// TwinCAT 3 PLC project Fraktal_Press_Demo
// Title: Fraktal_Press_Demo
// Company: fraktal-automation
// Author: fraktal-automation
// ProjectVersion: 0.1.0.9
// Description: CX2030 virtual/physical commissioning example: XTI-linked EK1200/EL1809/EL2809 HAL mapping, two-hand start, interlocked door/part slide, safety aliases, Control On/Off, AUTO/HOME/MANUAL, and model recipes.
// ProgramVersion: 3.1.4026.24
// libraries:
//   Fraktal_Core, 0.1.0.5 (fraktal-automation)
//   Fraktal_Modules, 0.1.0.4 (fraktal-automation)
//   Tc2_EtherCAT, * (Beckhoff Automation GmbH)
//   Tc2_Standard, * (Beckhoff Automation GmbH)
//   Tc2_System, * (Beckhoff Automation GmbH)
//   Tc3_Module, * (Beckhoff Automation GmbH)
// project tree:
//   00_System/Hardware/ GVL_PressIO.TcGVL, GVL_PressSafety.TcGVL (not stored)
//   / PlcTask.TcTTO (not stored)
//   01_PneumaticPress/Sequences/ FB_PressDemoLoadPosition.TcPOU, FB_PressDemoHome.TcPOU, FB_PressDemoChangeover.TcPOU, FB_PressDemoAuto.TcPOU
//   01_PneumaticPress/Release/ FB_PressDemoRelease.TcPOU (not stored)
//   01_PneumaticPress/ FB_PressDemoUnit.TcPOU
//   00_System/ MAIN.TcPOU, FB_PressIoDriver.TcPOU, FB_PressControlOnCircuit.TcPOU, FB_PressControlDomain.TcPOU, FB_PressOutputAuthority.TcPOU (not stored), FB_PressSimulationDriver.TcPOU (not stored)
//   01_PneumaticPress/Recipes/ FB_PressRecipeCatalog.TcPOU (not stored)
//   01_PneumaticPress/Io/ FB_PressIoCatalog.TcPOU (not stored), GVL_PressFieldbus.TcGVL (not stored)
// real-time tasks:
//   TASK PlcTask: cycle T#10ms, priority 20, ADS port 350
// I/O:
//   DEVICE =000+S-A610-A1 (EtherCAT), AmsNetId 0.0.0.0.2.1
//     =000+S-K010 (EK1200) [EK1200-5000 EtherCAT Power supply (2A E-Bus)]
//       =000+S-K010B1 (EL1809) [EL1809 16Ch. Dig. Input 24V, 3ms]
//       =000+S-K010C1 (EL2809) [EL2809 16Ch. Dig. Output 24V, 0.5A]
//       =000+S-K010D1 (EL6001) [EL6001 Interface (RS232)]
//       =000+S-K010E (EL9011) [EL9011 End Terminal]
// variable links:
//   Fraktal_Press_Demo/Fraktal_Press_Demo Instance <-> =000+S-A610-A1 (EtherCAT)/=000+S-K010 (EK1200)/=000+S-K010B1 (EL1809)
//     PlcTask Inputs/GVL_PressIO._000K910A <-> Channel 15/_000K910A
//     PlcTask Inputs/GVL_PressIO._000K911_Y32 <-> Channel 14/_000K911_Y32
//     PlcTask Inputs/GVL_PressIO._000MB085A_2 <-> Channel 10/_000MB085A_2
//     PlcTask Inputs/GVL_PressIO._000MB085A_4 <-> Channel 11/_000MB085A_4
//     PlcTask Inputs/GVL_PressIO._101B201A <-> Channel 3/_101B201A
//     PlcTask Inputs/GVL_PressIO._101B202A <-> Channel 5/_101B202A
//     PlcTask Inputs/GVL_PressIO._101B301A <-> Channel 1/_101B301A
//     PlcTask Inputs/GVL_PressIO._101B201B <-> Channel 4/_101B201B
//     PlcTask Inputs/GVL_PressIO._101B202B <-> Channel 6/_101B202B
//     PlcTask Inputs/GVL_PressIO._101B301B <-> Channel 2/_101B301B
//     PlcTask Inputs/GVL_PressIO._101B601 <-> Channel 12/_101B601
//     PlcTask Inputs/GVL_PressIO._101S101 <-> Channel 7/_101S101
//     PlcTask Inputs/GVL_PressIO._101S102 <-> Channel 8/_101S102
//   Fraktal_Press_Demo/Fraktal_Press_Demo Instance <-> =000+S-A610-A1 (EtherCAT)/=000+S-K010 (EK1200)/=000+S-K010C1 (EL2809)
//     PlcTask Outputs/GVL_PressIO._000K911_A1 <-> Channel 11/_000K911_A1
//     PlcTask Outputs/GVL_PressIO._000K951_A1 <-> Channel 10/_000K951_A1
//     PlcTask Outputs/GVL_PressIO._101K201A <-> Channel 3/_101K201A
//     PlcTask Outputs/GVL_PressIO._101K202A <-> Channel 5/_101K202A
//     PlcTask Outputs/GVL_PressIO._101K301A <-> Channel 1/_101K301A
//     PlcTask Outputs/GVL_PressIO._101K201B <-> Channel 4/_101K201B
//     PlcTask Outputs/GVL_PressIO._101K202B <-> Channel 6/_101K202B
//     PlcTask Outputs/GVL_PressIO._101K301B <-> Channel 2/_101K301B
//     PlcTask Outputs/GVL_PressIO._101P101 <-> Channel 7/_101P101
//     PlcTask Outputs/GVL_PressIO._101P102 <-> Channel 8/_101P102

// ---- 00_System/Hardware/GVL_PressIO.TcGVL
{attribute 'qualified_only'}
// CX2030 local EtherCAT process image, reconciled with the supplied XTI export.
// TcLinkTo owns the physical link by exact terminal/channel/PDO-entry name;
// AT %I*/%Q* keeps the compiler-selected process-image offset non-positional.
VAR_GLOBAL
    // =000+S-K010B1 (EL1809) inputs
    {attribute 'TcLinkTo' := 'TIIB[=000+S-K010B1 (EL1809)]^Channel 1^_101B301A'}
    _101B301A AT %I* : BOOL;       // Ch1 feeder retracted = logical slide INSIDE
    {attribute 'TcLinkTo' := 'TIIB[=000+S-K010B1 (EL1809)]^Channel 2^_101B301B'}
    _101B301B AT %I* : BOOL;       // Ch2 feeder extended  = logical slide OUTSIDE
    {attribute 'TcLinkTo' := 'TIIB[=000+S-K010B1 (EL1809)]^Channel 3^_101B201A'}
    _101B201A AT %I* : BOOL;       // Ch3 door closed
    {attribute 'TcLinkTo' := 'TIIB[=000+S-K010B1 (EL1809)]^Channel 4^_101B201B'}
    _101B201B AT %I* : BOOL;       // Ch4 door open
    {attribute 'TcLinkTo' := 'TIIB[=000+S-K010B1 (EL1809)]^Channel 5^_101B202A'}
    _101B202A AT %I* : BOOL;       // Ch5 press down
    {attribute 'TcLinkTo' := 'TIIB[=000+S-K010B1 (EL1809)]^Channel 6^_101B202B'}
    _101B202B AT %I* : BOOL;       // Ch6 press up
    {attribute 'TcLinkTo' := 'TIIB[=000+S-K010B1 (EL1809)]^Channel 7^_101S101'}
    _101S101  AT %I* : BOOL;       // Ch7 right two-hand raw button
    {attribute 'TcLinkTo' := 'TIIB[=000+S-K010B1 (EL1809)]^Channel 8^_101S102'}
    _101S102  AT %I* : BOOL;       // Ch8 left two-hand raw button
    {attribute 'TcLinkTo' := 'TIIB[=000+S-K010B1 (EL1809)]^Channel 10^_000MB085A_2'}
    _000MB085A_2 AT %I* : BOOL;    // Ch10 compressed air below 0.3 bar
    {attribute 'TcLinkTo' := 'TIIB[=000+S-K010B1 (EL1809)]^Channel 11^_000MB085A_4'}
    _000MB085A_4 AT %I* : BOOL;    // Ch11 compressed air above 4.5 bar
    {attribute 'TcLinkTo' := 'TIIB[=000+S-K010B1 (EL1809)]^Channel 12^_101B601'}
    _101B601 AT %I* : BOOL;        // Ch12 part present
    // N54 D2 operator buttons. Free EL1809 channels were 9/13/16; 9 and 13 are
    // assigned here. The TcLinkTo names MUST match the terminal channel names in
    // XAE - confirm the physical wiring before trusting these.
    {attribute 'TcLinkTo' := 'TIIB[=000+S-K010B1 (EL1809)]^Channel 9^_000BS901'}
    _000BS901 AT %I* : BOOL;       // Ch9  IsControlOnButtonPressed  (=000+B-S901:14)
    {attribute 'TcLinkTo' := 'TIIB[=000+S-K010B1 (EL1809)]^Channel 13^_000BS902'}
    _000BS902 AT %I* : BOOL;       // Ch13 IsControlOffButtonPressed (=000+B-S902:14)
    {attribute 'TcLinkTo' := 'TIIB[=000+S-K010B1 (EL1809)]^Channel 14^_000K911_Y32'}
    _000K911_Y32 AT %I* : BOOL;    // Ch14 Control On feedback
    {attribute 'TcLinkTo' := 'TIIB[=000+S-K010B1 (EL1809)]^Channel 15^_000K910A'}
    _000K910A AT %I* : BOOL;       // Ch15 E-stop PRESSED (=000+S1-K910A:14); NORMALLY OPEN on this
                                   // demo rig: TRUE = actuated. NOT fail-safe - production needs NC.

    // =000+S-K010C1 (EL2809) outputs
    {attribute 'TcLinkTo' := 'TIIB[=000+S-K010C1 (EL2809)]^Channel 1^_101K301A'}
    _101K301A AT %Q* : BOOL;       // Ch1 feeder backward = move inside
    {attribute 'TcLinkTo' := 'TIIB[=000+S-K010C1 (EL2809)]^Channel 2^_101K301B'}
    _101K301B AT %Q* : BOOL;       // Ch2 feeder forward  = move outside
    {attribute 'TcLinkTo' := 'TIIB[=000+S-K010C1 (EL2809)]^Channel 3^_101K201A'}
    _101K201A AT %Q* : BOOL;       // Ch3 close door
    {attribute 'TcLinkTo' := 'TIIB[=000+S-K010C1 (EL2809)]^Channel 4^_101K201B'}
    _101K201B AT %Q* : BOOL;       // Ch4 open door
    {attribute 'TcLinkTo' := 'TIIB[=000+S-K010C1 (EL2809)]^Channel 5^_101K202A'}
    _101K202A AT %Q* : BOOL;       // Ch5 press downward
    {attribute 'TcLinkTo' := 'TIIB[=000+S-K010C1 (EL2809)]^Channel 6^_101K202B'}
    _101K202B AT %Q* : BOOL;       // Ch6 press upward
    {attribute 'TcLinkTo' := 'TIIB[=000+S-K010C1 (EL2809)]^Channel 7^_101P101'}
    _101P101  AT %Q* : BOOL;       // Ch7 right two-hand lamp
    {attribute 'TcLinkTo' := 'TIIB[=000+S-K010C1 (EL2809)]^Channel 8^_101P102'}
    _101P102  AT %Q* : BOOL;       // Ch8 left two-hand lamp
    {attribute 'TcLinkTo' := 'TIIB[=000+S-K010C1 (EL2809)]^Channel 10^_000K951_A1'}
    _000K951_A1 AT %Q* : BOOL;     // Ch10 SwitchControlOn functional request
    {attribute 'TcLinkTo' := 'TIIB[=000+S-K010C1 (EL2809)]^Channel 11^_000K911_A1'}
    _000K911_A1 AT %Q* : BOOL;     // Ch11 EnableControlOn functional request
END_VAR

// ---- 01_PneumaticPress/Sequences/FB_PressDemoLoadPosition.TcPOU
// Shared load-safe-position sub-sequence (Core §6.7): ram up, door open, slide
// outside. HOME and CHANGEOVER both embed it as one composite step, passing a
// BaseStepNo window so its detailed progress projects through the Unit's normal
// §6.5 step record. Implemented as a Core §6.8 ST `CASE _step OF` skeleton on
// FB_SequenceBase — the step actions issue child commands only through the §6.1
// handshake (M_MayIssue), and progression rides the shared _retVal via M_Advance.
FUNCTION_BLOCK FB_PressDemoLoadPosition EXTENDS FB_SequenceBase
VAR
    _baseStepNo : INT;
    {attribute 'OPC.UA.DA' := '0'}
    _pressRam : REFERENCE TO FB_CylinderCM;
    {attribute 'OPC.UA.DA' := '0'}
    _door : REFERENCE TO FB_CylinderCM;
    {attribute 'OPC.UA.DA' := '0'}
    _partSlide : REFERENCE TO FB_CylinderCM;
END_VAR

// step body runs via M_Run; the Unit calls this instance each scan

METHOD M_Reset
VAR_INPUT
    BaseStepNo : INT;
END_VAR
_baseStepNo := BaseStepNo;
M_ResetBase();
END_METHOD

// §6.8 ST step skeleton. One M_Step per step, one commit via M_Advance.
METHOD M_Run
IF NOT _attached THEN
    RETURN;
END_IF
CASE _step OF
    0:  // ram up
        M_Step(StepNo := _baseStepNo, StepName := 'project.step.pressSafePositionRamUp',
            Awaits := _pressRam, AwaitingLabel := 'PressRam.RETRACT',
            TimeClass := E_TimeClass.WORK, ExpectedTime := T#0S);
        IF M_MayIssue(Steppable := TRUE) THEN
            _pressRam.Abort := FALSE;
            _pressRam.Command := E_CylinderCommand.RETRACT;
            _pressRam.Execute := TRUE;
        END_IF
        IF _pressRam.Done THEN
            _pressRam.Execute := FALSE;
            _retVal := E_StepResult.ADVANCE;
        END_IF
        M_Advance(OnAdvance := 20);
    20:  // door open
        M_Step(StepNo := _baseStepNo + 20, StepName := 'project.step.pressSafePositionDoorOpen',
            Awaits := _door, AwaitingLabel := 'Door.RETRACT',
            TimeClass := E_TimeClass.WORK, ExpectedTime := T#0S);
        IF M_MayIssue(Steppable := TRUE) THEN
            _door.Abort := FALSE;
            _door.Command := E_CylinderCommand.RETRACT;
            _door.Execute := TRUE;
        END_IF
        IF _door.Done THEN
            _door.Execute := FALSE;
            _retVal := E_StepResult.ADVANCE;
        END_IF
        M_Advance(OnAdvance := 40);
    40:  // slide outside
        M_Step(StepNo := _baseStepNo + 40, StepName := 'project.step.pressSafePositionSlideOutside',
            Awaits := _partSlide, AwaitingLabel := 'PartSlide.RETRACT',
            TimeClass := E_TimeClass.WORK, ExpectedTime := T#0S);
        IF M_MayIssue(Steppable := TRUE) THEN
            _partSlide.Abort := FALSE;
            _partSlide.Command := E_CylinderCommand.RETRACT;
            _partSlide.Execute := TRUE;
        END_IF
        IF _partSlide.Done THEN
            _partSlide.Execute := FALSE;
            _retVal := E_StepResult.ADVANCE;
        END_IF
        M_Advance(OnAdvance := 999);
    999:  // established
        M_Step(StepNo := _baseStepNo + 60, StepName := 'project.step.pressSafePositionComplete',
            Awaits := 0, AwaitingLabel := '', TimeClass := E_TimeClass.WORK, ExpectedTime := T#0S);
        Done := TRUE;
ELSE
    M_Fault(Reason := E_Reason.STEP_STALLED, DescriptionKey := 'std.error.undefinedStep');
END_CASE
END_METHOD

METHOD Setup : BOOL
VAR_INPUT
    Host : I_SequenceHost;
END_VAR
VAR_IN_OUT
    PressRam : FB_CylinderCM;
    Door : FB_CylinderCM;
    PartSlide : FB_CylinderCM;
END_VAR
_pressRam REF= PressRam;
_door REF= Door;
_partSlide REF= PartSlide;
Setup := M_Attach(Host := Host)
    AND __ISVALIDREF(_pressRam) AND __ISVALIDREF(_door) AND __ISVALIDREF(_partSlide);
END_METHOD

END_FUNCTION_BLOCK

// ---- 01_PneumaticPress/Sequences/FB_PressDemoHome.TcPOU
// HOME mode chain (Core §6.2/§6.8 ST skeleton on FB_SequenceBase): establish the
// shared load-safe position, then complete. Finite (does not loop).
FUNCTION_BLOCK FB_PressDemoHome EXTENDS FB_SequenceBase
VAR
    {attribute 'OPC.UA.DA' := '0'}
    _outCmd : REFERENCE TO ST_PneumaticPressOutCmd;
    {attribute 'OPC.UA.DA' := '0'}
    _loadPosition : FB_PressDemoLoadPosition;
    _loadPositionRunning : BOOL;
END_VAR

METHOD M_Reset
M_ResetBase();
_loadPositionRunning := FALSE;
_loadPosition.M_Reset(BaseStepNo := 0);
END_METHOD

METHOD M_Run
IF NOT _attached THEN
    RETURN;
END_IF
CASE _step OF
    0:  // initialize
        M_Step(StepNo := 0, StepName := 'project.step.pressHomeInitialize',
            Awaits := 0, AwaitingLabel := '', TimeClass := E_TimeClass.WORK, ExpectedTime := T#0S);
        _outCmd.Homed := FALSE;
        _outCmd.ChangeoverCompleted := FALSE;
        _loadPositionRunning := FALSE;
        _retVal := E_StepResult.ADVANCE;
        M_Advance(OnAdvance := 900);
    900:  // shared load-safe position (composite step, §6.7)
        IF NOT _loadPositionRunning THEN
            _loadPosition.M_Reset(BaseStepNo := 900);
            _loadPositionRunning := TRUE;
        END_IF
        _loadPosition.M_Run();
        IF _loadPosition.Done THEN
            _loadPositionRunning := FALSE;
            _retVal := E_StepResult.ADVANCE;
        END_IF
        M_Advance(OnAdvance := 999);
    999:  // complete
        M_Step(StepNo := 999, StepName := 'project.step.pressHomeComplete',
            Awaits := 0, AwaitingLabel := '', TimeClass := E_TimeClass.WORK, ExpectedTime := T#0S);
        _outCmd.Homed := TRUE;
        M_Complete();
ELSE
    M_Fault(Reason := E_Reason.STEP_STALLED, DescriptionKey := 'std.error.undefinedStep');
END_CASE
END_METHOD

METHOD Setup : BOOL
VAR_INPUT
    Host : I_SequenceHost;
END_VAR
VAR_IN_OUT
    PressRam : FB_CylinderCM;
    Door : FB_CylinderCM;
    PartSlide : FB_CylinderCM;
    OutCmd : ST_PneumaticPressOutCmd;
END_VAR
_outCmd REF= OutCmd;
Setup := M_Attach(Host := Host) AND __ISVALIDREF(_outCmd)
    AND _loadPosition.Setup(Host := Host, PressRam := PressRam, Door := Door, PartSlide := PartSlide);
END_METHOD

END_FUNCTION_BLOCK

// ---- 01_PneumaticPress/Sequences/FB_PressDemoChangeover.TcPOU
// CHANGEOVER mode chain (Core §6.2/§6.8 ST skeleton on FB_SequenceBase): validate
// the selected model, establish the shared load-safe position, then ask the
// operator (§6.11) to confirm tooling/material match before completing. The
// 'repeat position' answer restarts the guided move via a backward jump (§6.10).
FUNCTION_BLOCK FB_PressDemoChangeover EXTENDS FB_SequenceBase
VAR
    _decisionRequest : ST_DecisionRequest;
    _answer : INT;
    _modelSelected : BOOL;
    {attribute 'OPC.UA.DA' := '0'}
    _outCmd : REFERENCE TO ST_PneumaticPressOutCmd;
    {attribute 'OPC.UA.DA' := '0'}
    _model : REFERENCE TO ST_ModelId;
    {attribute 'OPC.UA.DA' := '0'}
    _loadPosition : FB_PressDemoLoadPosition;
    _loadPositionRunning : BOOL;
END_VAR

METHOD M_Reset
M_ResetBase();
_answer := 0;
_loadPositionRunning := FALSE;
_loadPosition.M_Reset(BaseStepNo := 0);
END_METHOD

METHOD M_Run
IF NOT _attached THEN
    RETURN;
END_IF
CASE _step OF
    0:  // initialize
        M_Step(StepNo := 0, StepName := 'project.step.pressChangeoverInitialize',
            Awaits := 0, AwaitingLabel := '', TimeClass := E_TimeClass.WORK, ExpectedTime := T#0S);
        _outCmd.ChangeoverCompleted := FALSE;
        _outCmd.Homed := FALSE;
        _answer := 0;
        _decisionRequest.Prompt := '';
        M_ClearDecision();
        _loadPositionRunning := FALSE;
        _retVal := E_StepResult.ADVANCE;
        M_Advance(OnAdvance := 800);
    800:  // validate the transactionally-loaded model
        M_Step(StepNo := 800, StepName := 'project.step.pressChangeoverValidateModel',
            Awaits := 0, AwaitingLabel := '', TimeClass := E_TimeClass.WAIT_OPERATOR, ExpectedTime := T#0S);
        _modelSelected := M_Await(Idx := 1, Label := 'project.condition.pressModelSelected',
            Ok := _model.ModelCode <> '');
        IF _modelSelected THEN
            _loadPositionRunning := FALSE;
            _retVal := E_StepResult.ADVANCE;
        END_IF
        M_Advance(OnAdvance := 810);
    810:  // shared load-safe position (composite step)
        IF NOT _loadPositionRunning THEN
            _loadPosition.M_Reset(BaseStepNo := 810);
            _loadPositionRunning := TRUE;
        END_IF
        _loadPosition.M_Run();
        IF _loadPosition.Done THEN
            _loadPositionRunning := FALSE;
            _retVal := E_StepResult.ADVANCE;
        END_IF
        M_Advance(OnAdvance := 870);
    870:  // request tooling/material confirmation
        M_Step(StepNo := 870, StepName := 'project.step.pressChangeoverRequestConfirmation',
            Awaits := 0, AwaitingLabel := '', TimeClass := E_TimeClass.WAIT_OPERATOR, ExpectedTime := T#0S);
        _decisionRequest.Prompt := 'project.decision.pressChangeoverConfirm';
        _decisionRequest.Options[1] := 'project.decision.confirmChangeover';
        _decisionRequest.Options[2] := 'project.decision.repeatChangeoverPosition';
        _decisionRequest.Default := 0;
        _decisionRequest.Timeout := T#0S;
        M_AskDecision(Req := _decisionRequest);
        _retVal := E_StepResult.ADVANCE;
        M_Advance(OnAdvance := 880);
    880:  // await confirmation; JUMP1 = repeat the guided position
        M_Step(StepNo := 880, StepName := 'project.step.pressChangeoverAwaitConfirmation',
            Awaits := 0, AwaitingLabel := '', TimeClass := E_TimeClass.WAIT_OPERATOR, ExpectedTime := T#0S);
        _answer := M_TakeDecision();
        IF _answer = 1 THEN
            _retVal := E_StepResult.ADVANCE;
        ELSIF _answer = 2 THEN
            _loadPositionRunning := FALSE;      // repeat the guided position from the start
            _retVal := E_StepResult.JUMP1;
        ELSE
            _modelSelected := M_Await(Idx := 1,
                Label := 'project.condition.pressChangeoverConfirmation', Ok := FALSE);
        END_IF
        M_Advance(OnAdvance := 999, OnJump1 := 810);
    999:  // complete
        M_Step(StepNo := 999, StepName := 'project.step.pressChangeoverComplete',
            Awaits := 0, AwaitingLabel := '', TimeClass := E_TimeClass.WORK, ExpectedTime := T#0S);
        _outCmd.Homed := TRUE;
        _outCmd.ChangeoverCompleted := TRUE;
        M_Complete();
ELSE
    M_Fault(Reason := E_Reason.STEP_STALLED, DescriptionKey := 'std.error.undefinedStep');
END_CASE
END_METHOD

METHOD Setup : BOOL
VAR_INPUT
    Host : I_SequenceHost;
END_VAR
VAR_IN_OUT
    PressRam : FB_CylinderCM;
    Door : FB_CylinderCM;
    PartSlide : FB_CylinderCM;
    OutCmd : ST_PneumaticPressOutCmd;
    Model : ST_ModelId;
END_VAR
_outCmd REF= OutCmd;
_model REF= Model;
Setup := M_Attach(Host := Host) AND __ISVALIDREF(_outCmd) AND __ISVALIDREF(_model)
    AND _loadPosition.Setup(Host := Host, PressRam := PressRam, Door := Door, PartSlide := PartSlide);
END_METHOD

END_FUNCTION_BLOCK

// ---- 01_PneumaticPress/Sequences/FB_PressDemoAuto.TcPOU
// AUTO mode chain (Core §6.2/§6.8 ST skeleton on FB_SequenceBase): the continuous
// production cycle — await a fresh two-hand start with part+air present, transfer
// the part in, press for the recipe dwell, return to load position, count the good
// part, and loop until Stop. A Stop requested at the between-cycles wait is honored
// there (M_StopNow) so no phantom cycle is charged. Every child motion goes through
// the §6.1 handshake (M_MayIssue); progression rides the shared _retVal.
FUNCTION_BLOCK FB_PressDemoAuto EXTENDS FB_SequenceBase
VAR
    _partReady, _airReady, _startReady : BOOL;
    _traceAccepted, _recordAccepted, _partProcessed : BOOL;
    {attribute 'OPC.UA.DA' := '0'}
    _pressRam : REFERENCE TO FB_CylinderCM;
    {attribute 'OPC.UA.DA' := '0'}
    _door : REFERENCE TO FB_CylinderCM;
    {attribute 'OPC.UA.DA' := '0'}
    _partSlide : REFERENCE TO FB_CylinderCM;
    {attribute 'OPC.UA.DA' := '0'}
    _twoHand : REFERENCE TO FB_TwoHandStartCM;
    {attribute 'OPC.UA.DA' := '0'}
    _partPresentSensor : REFERENCE TO FB_DigitalInputCM;
    {attribute 'OPC.UA.DA' := '0'}
    _airPressureMonitor : REFERENCE TO FB_AirPressureMonitorCM;
    {attribute 'OPC.UA.DA' := '0'}
    _parCfg : REFERENCE TO ST_PneumaticPressParCfg;
    {attribute 'OPC.UA.DA' := '0'}
    _outCmd : REFERENCE TO ST_PneumaticPressOutCmd;
    {attribute 'OPC.UA.DA' := '0'}
    _startLatched : REFERENCE TO BOOL;
    {attribute 'OPC.UA.DA' := '0'}
    _loadPosition : FB_PressDemoLoadPosition;
    _loadPositionRunning : BOOL;
END_VAR

METHOD M_Reset
M_ResetBase(0);
_loadPositionRunning := FALSE;
_loadPosition.M_Reset(BaseStepNo := 0);
END_METHOD

METHOD M_Run
IF NOT _attached THEN
    RETURN;
END_IF
CASE _step OF
    0:  // initialize
        M_Step(StepNo := 0, StepName := 'project.step.pressAutoInitialize',
            Awaits := 0, AwaitingLabel := '', TimeClass := E_TimeClass.WORK, ExpectedTime := T#0S);
        _outCmd.CycleCompleted := FALSE;
        _outCmd.Homed := FALSE;
        _outCmd.ChangeoverCompleted := FALSE;
        _loadPositionRunning := FALSE;
        _retVal := E_StepResult.ADVANCE;
        M_Advance(OnAdvance := 100, OnJump1 := -1, OnJump2 := -1, OnJump3 := -1);
    100:  // await a fresh two-hand start (the §8.11.1 cycle-start marker)
        M_Step(StepNo := 100, StepName := 'project.step.pressAwaitTwoHand',
            Awaits := 0, AwaitingLabel := '', TimeClass := E_TimeClass.WAIT_OPERATOR, ExpectedTime := T#0S);
        _outCmd.CycleCompleted := FALSE;
        _partReady := M_Await(Idx := 1, Label := 'project.condition.partPresent',
            Ok := _partPresentSensor.OutImm.Value AND _partPresentSensor.OutImm.Quality);
        _airReady := M_Await(Idx := 2, Label := 'project.condition.airPressureOk',
            Ok := _airPressureMonitor.OutImm.PressureOk);
        IF _parCfg.RequireTwoHandStart THEN
            _startReady := M_Await(Idx := 3, Label := 'project.condition.twoHandStart', Ok := _startLatched);
        ELSE
            _startReady := TRUE;
        END_IF
        IF M_StopPending() THEN
            M_StopNow();                       // stop accepted BETWEEN cycles: no phantom cycle
        ELSIF _partReady AND _airReady AND _startReady THEN
            _traceAccepted := M_PartReceived();
            _retVal := E_StepResult.ADVANCE;
        END_IF
        M_Advance(OnAdvance := 110, OnJump1 := -1, OnJump2 := -1, OnJump3 := -1);
    110:  // ram up
        M_Step(StepNo := 110, StepName := 'project.step.pressRamUp',
            Awaits := _pressRam, AwaitingLabel := 'PressRam.RETRACT', TimeClass := E_TimeClass.WORK, ExpectedTime := T#0S);
        IF M_MayIssue(Steppable := TRUE) THEN
            _pressRam.Abort := FALSE; _pressRam.Command := E_CylinderCommand.RETRACT; _pressRam.Execute := TRUE;
        END_IF
        IF _pressRam.Done THEN _pressRam.Execute := FALSE; _retVal := E_StepResult.ADVANCE; END_IF
        M_Advance(OnAdvance := 130, OnJump1 := -1, OnJump2 := -1, OnJump3 := -1);
    130:  // door open
        M_Step(StepNo := 130, StepName := 'project.step.pressDoorOpen',
            Awaits := _door, AwaitingLabel := 'Door.RETRACT', TimeClass := E_TimeClass.WORK, ExpectedTime := T#0S);
        IF M_MayIssue(Steppable := TRUE) THEN
            _door.Abort := FALSE; _door.Command := E_CylinderCommand.RETRACT; _door.Execute := TRUE;
        END_IF
        IF _door.Done THEN _door.Execute := FALSE; _retVal := E_StepResult.ADVANCE; END_IF
        M_Advance(OnAdvance := 150, OnJump1 := -1, OnJump2 := -1, OnJump3 := -1);
    150:  // slide inside (value-adding sequence begins)
        M_Step(StepNo := 150, StepName := 'project.step.pressSlideInside',
            Awaits := _partSlide, AwaitingLabel := 'PartSlide.EXTEND', TimeClass := E_TimeClass.WORK, ExpectedTime := T#0S);
        IF M_MayIssue(Steppable := TRUE) THEN
            M_PartStarted();
            _partSlide.Abort := FALSE; _partSlide.Command := E_CylinderCommand.EXTEND; _partSlide.Execute := TRUE;
        END_IF
        IF _partSlide.Done THEN _partSlide.Execute := FALSE; _retVal := E_StepResult.ADVANCE; END_IF
        M_Advance(OnAdvance := 170, OnJump1 := -1, OnJump2 := -1, OnJump3 := -1);
    170:  // transfer settle
        M_Step(StepNo := 170, StepName := 'project.step.pressTransferSettle',
            Awaits := 0, AwaitingLabel := '', TimeClass := E_TimeClass.WORK, ExpectedTime := _parCfg.TransferSettleTime);
        _retVal := M_Delay(PT := _parCfg.TransferSettleTime);
        M_Advance(OnAdvance := 180, OnJump1 := -1, OnJump2 := -1, OnJump3 := -1);
    180:  // door close
        M_Step(StepNo := 180, StepName := 'project.step.pressDoorClose',
            Awaits := _door, AwaitingLabel := 'Door.EXTEND', TimeClass := E_TimeClass.WORK, ExpectedTime := T#0S);
        IF M_MayIssue(Steppable := TRUE) THEN
            _door.Abort := FALSE; _door.Command := E_CylinderCommand.EXTEND; _door.Execute := TRUE;
        END_IF
        IF _door.Done THEN _door.Execute := FALSE; _retVal := E_StepResult.ADVANCE; END_IF
        M_Advance(OnAdvance := 200, OnJump1 := -1, OnJump2 := -1, OnJump3 := -1);
    200:  // ram down
        M_Step(StepNo := 200, StepName := 'project.step.pressRamDown',
            Awaits := _pressRam, AwaitingLabel := 'PressRam.EXTEND', TimeClass := E_TimeClass.WORK, ExpectedTime := T#0S);
        IF M_MayIssue(Steppable := TRUE) THEN
            _pressRam.Abort := FALSE; _pressRam.Command := E_CylinderCommand.EXTEND; _pressRam.Execute := TRUE;
        END_IF
        IF _pressRam.Done THEN _pressRam.Execute := FALSE; _retVal := E_StepResult.ADVANCE; END_IF
        M_Advance(OnAdvance := 220, OnJump1 := -1, OnJump2 := -1, OnJump3 := -1);
    220:  // press dwell — two-hand must stay active
        M_Step(StepNo := 220, StepName := 'project.step.pressDwell',
            Awaits := 0, AwaitingLabel := '', TimeClass := E_TimeClass.WORK, ExpectedTime := _parCfg.PressSettleTime);
        IF NOT _twoHand.OutImm.SafeActive AND _parCfg.RequireTwoHandStart THEN
            _pressRam.WithdrawOutputs();
            M_Fault(Reason := E_Reason.INTERLOCK_DROPPED, DescriptionKey := 'project.error.twoHandReleasedDuringPress');
        ELSE
            _retVal := M_Delay(PT := _parCfg.PressSettleTime);
        END_IF
        M_Advance(OnAdvance := 230, OnJump1 := -1, OnJump2 := -1, OnJump3 := -1);
    230:  // record the applied dwell (§3.16.1 measured value)
        M_Step(StepNo := 230, StepName := 'project.step.pressRecordResult',
            Awaits := 0, AwaitingLabel := '', TimeClass := E_TimeClass.WORK, ExpectedTime := T#0S);
        _recordAccepted := M_PartRecord(RecordName := 'PressDwell',
            Value := DINT_TO_LREAL(TIME_TO_DINT(_parCfg.PressSettleTime)),
            Minimum := 0, Maximum := 30000,
            Target := DINT_TO_LREAL(TIME_TO_DINT(_parCfg.PressSettleTime)), EngUnit := 'ms');
        _loadPositionRunning := FALSE;
        _retVal := E_StepResult.ADVANCE;
        M_Advance(OnAdvance := 240, OnJump1 := -1, OnJump2 := -1, OnJump3 := -1);
    240:  // return to the shared load-safe position (composite step)
        IF NOT _loadPositionRunning THEN
            _loadPosition.M_Reset(BaseStepNo := 240);
            _loadPositionRunning := TRUE;
        END_IF
        _loadPosition.M_Run();
        IF _loadPosition.Done THEN
            _loadPositionRunning := FALSE;
            _retVal := E_StepResult.ADVANCE;
        END_IF
        M_Advance(OnAdvance := 999, OnJump1 := -1, OnJump2 := -1, OnJump3 := -1);
    999:  // cycle complete — write result, count by verdict, loop (§8.11.1 finish marker)
        M_Step(StepNo := 999, StepName := 'project.step.pressAutoComplete',
            Awaits := 0, AwaitingLabel := '', TimeClass := E_TimeClass.WORK, ExpectedTime := T#0S);
        _outCmd.CycleCompleted := TRUE;
        _partProcessed := M_PartProcessed(Verdict := E_Verdict.OK, Reason := E_Reason.NONE);
        IF NOT _partProcessed THEN
            M_CountGood();                     // §3.9: no carrier configured — count directly
        END_IF
        _startLatched := FALSE;
        IF M_EndOfCycle() THEN
            _retVal := E_StepResult.ADVANCE;   // stop NOT requested: loop to N100
        END_IF
        M_Advance(OnAdvance := 100, OnJump1 := -1, OnJump2 := -1, OnJump3 := -1);
ELSE
    M_Fault(Reason := E_Reason.STEP_STALLED, DescriptionKey := 'std.error.undefinedStep');
END_CASE
END_METHOD

METHOD Setup : BOOL
VAR_INPUT
    Host : I_SequenceHost;
END_VAR
VAR_IN_OUT
    PressRam : FB_CylinderCM;
    Door : FB_CylinderCM;
    PartSlide : FB_CylinderCM;
    TwoHand : FB_TwoHandStartCM;
    PartPresentSensor : FB_DigitalInputCM;
    AirPressureMonitor : FB_AirPressureMonitorCM;
    ParCfg : ST_PneumaticPressParCfg;
    OutCmd : ST_PneumaticPressOutCmd;
    StartLatched : BOOL;
END_VAR
_pressRam REF= PressRam;
_door REF= Door;
_partSlide REF= PartSlide;
_twoHand REF= TwoHand;
_partPresentSensor REF= PartPresentSensor;
_airPressureMonitor REF= AirPressureMonitor;
_parCfg REF= ParCfg;
_outCmd REF= OutCmd;
_startLatched REF= StartLatched;
Setup := M_Attach(Host := Host) AND __ISVALIDREF(_pressRam) AND __ISVALIDREF(_door)
    AND __ISVALIDREF(_partSlide) AND __ISVALIDREF(_twoHand)
    AND __ISVALIDREF(_partPresentSensor) AND __ISVALIDREF(_airPressureMonitor)
    AND __ISVALIDREF(_parCfg) AND __ISVALIDREF(_outCmd) AND __ISVALIDREF(_startLatched)
    AND _loadPosition.Setup(Host := Host, PressRam := PressRam, Door := Door, PartSlide := PartSlide);
END_METHOD

END_FUNCTION_BLOCK

// ---- 01_PneumaticPress/FB_PressDemoUnit.TcPOU
// Project-owned Unit: pneumatic press + access door + transfer slide + two-hand request.
// Cylinder interlocks prevent the two documented collisions in AUTO and MANUAL.
// Certified E-stop, two-hand evaluation and safe valve outputs remain external.
FUNCTION_BLOCK FB_PressDemoUnit EXTENDS FB_UnitBase
VAR_INPUT
    ParCfg : ST_PneumaticPressParCfg;
    ParCmd : ST_PneumaticPressParCmd;
END_VAR
VAR_OUTPUT
    PressRam      : FB_CylinderCM;
    Door          : FB_CylinderCM;
    PartSlide     : FB_CylinderCM;
    TwoHand       : FB_TwoHandStartCM;
    PneumaticPower: FB_PowerGroupCM;
    PartPresentSensor : FB_DigitalInputCM;
    AirPressureMonitor : FB_AirPressureMonitorCM;
    ReleaseConditions : FB_PressDemoRelease; // project-owned, browseable condition state
    OutCmd        : ST_PneumaticPressOutCmd;
    OutImm        : ST_PneumaticPressOutImm;
END_VAR
VAR
    {attribute 'OPC.UA.DA' := '0'}
    _recipe : I_RecipeProvider;
    _parCfgStaged : ST_PneumaticPressParCfg;
    _recipePrepared : BOOL;
    _startLatched : BOOL;
    _powerRequestPending : BOOL;
    _powerTargetOn : BOOL;
    {attribute 'OPC.UA.DA' := '0'}
    _homeSequence : FB_PressDemoHome;       // §6.8 ST chain on FB_SequenceBase owns HOME steps
    {attribute 'OPC.UA.DA' := '0'}
    _changeoverSequence : FB_PressDemoChangeover;
    {attribute 'OPC.UA.DA' := '0'}
    _autoSequence : FB_PressDemoAuto;
END_VAR

Cyclic();

METHOD Setup : BOOL
VAR_INPUT
    Name : STRING(80);
    PressHal : REFERENCE TO ST_CylinderHal;
    DoorHal : REFERENCE TO ST_CylinderHal;
    SlideHal : REFERENCE TO ST_CylinderHal;
    TwoHandHal : REFERENCE TO ST_TwoHandHal;
    PowerHal : REFERENCE TO ST_PowerGroupHal;
    PartPresentHal : REFERENCE TO ST_DigitalInputHal;
    AirPressureHal : REFERENCE TO ST_AirPressureHal;
    Recipe : I_RecipeProvider;
END_VAR
VAR
    InitialModel : ST_ModelId;
    Ok : BOOL;
END_VAR
_M_SetName(Name);
_M_SetPresentation(DisplayNameKey := 'project.module.pneumaticPress.name', DescriptionKey := 'project.module.pneumaticPress.description');
_recipe := Recipe;
Ok := PressRam.Setup(Name := CONCAT(Name, '.PressRam'), HalRef := PressHal, Recipe := 0);
Ok := Door.Setup(Name := CONCAT(Name, '.Door'), HalRef := DoorHal, Recipe := 0) AND Ok;
Ok := PartSlide.Setup(Name := CONCAT(Name, '.PartSlide'), HalRef := SlideHal, Recipe := 0) AND Ok;
Ok := TwoHand.Setup(Name := CONCAT(Name, '.TwoHand'), HalRef := TwoHandHal) AND Ok;
Ok := PneumaticPower.Setup(Name := CONCAT(Name, '.PneumaticPower'), HalRef := PowerHal) AND Ok;
Ok := PartPresentSensor.Setup(Name := CONCAT(Name, '.PartPresentSensor'),
    HalRef := PartPresentHal, DisplayNameKey := 'project.module.partPresentSensor.name',
    DescriptionKey := 'project.module.partPresentSensor.description') AND Ok;
Ok := AirPressureMonitor.Setup(Name := CONCAT(Name, '.AirPressureMonitor'),
    HalRef := AirPressureHal) AND Ok;
Ok := ReleaseConditions.Setup(UnitPath := Name) AND Ok;
Ok := _homeSequence.Setup(Host := THIS^, PressRam := PressRam, Door := Door,
    PartSlide := PartSlide, OutCmd := OutCmd) AND Ok;
Ok := _changeoverSequence.Setup(Host := THIS^, PressRam := PressRam, Door := Door,
    PartSlide := PartSlide, OutCmd := OutCmd, Model := Model) AND Ok;
Ok := _autoSequence.Setup(Host := THIS^, PressRam := PressRam, Door := Door,
    PartSlide := PartSlide, TwoHand := TwoHand, PartPresentSensor := PartPresentSensor,
    AirPressureMonitor := AirPressureMonitor, ParCfg := ParCfg, OutCmd := OutCmd,
    StartLatched := _startLatched) AND Ok;
PneumaticPower.ParCfg.Kind := E_PowerGroupKind.VALVE_ZONE;
PneumaticPower.ParCfg.RequiredForControl := TRUE;
PneumaticPower.ParCfg.FieldbusLossReaction := E_FieldbusLossReaction.CONTROL_OFF;
Ok := _M_Register(PressRam) AND Ok;
Ok := _M_Register(Door) AND Ok;
Ok := _M_Register(PartSlide) AND Ok;
Ok := _M_Register(TwoHand) AND Ok;
Ok := _M_Register(PneumaticPower) AND Ok;
Ok := _M_Register(PartPresentSensor) AND Ok;
Ok := _M_Register(AirPressureMonitor) AND Ok;
Setup := Ok AND PrepareRecipe(Model := InitialModel);
IF Setup THEN CommitRecipe(); END_IF
END_METHOD

METHOD PrepareRecipe : BOOL
VAR_INPUT
    Model : ST_ModelId;
END_VAR
IF _recipe = 0 THEN
    _parCfgStaged := ParCfg;
    _recipePrepared := TRUE;
ELSIF _recipe.Load(ModelCode := Model.ModelCode, RecipeKey := 'PneumaticPressUnit', pParCfg := ADR(_parCfgStaged), Size := SIZEOF(_parCfgStaged)) THEN
    IF (_parCfgStaged.PressSettleTime > T#30S) OR (_parCfgStaged.TransferSettleTime > T#5S) THEN
        _M_Fault(E_Reason.RECIPE_INVALID, 'project.error.pressRecipeInvalid');
        _recipePrepared := FALSE;
        PrepareRecipe := FALSE;
        RETURN;
    END_IF
    _recipePrepared := TRUE;
ELSE
    _M_Fault(E_Reason.RECIPE_INVALID, 'std.error.recipeSchemaInvalid');
    _recipePrepared := FALSE;
    PrepareRecipe := FALSE;
    RETURN;
END_IF
PrepareRecipe := SUPER^.PrepareRecipe(Model := Model);
IF NOT PrepareRecipe THEN _recipePrepared := FALSE; END_IF
END_METHOD

METHOD CommitRecipe
SUPER^.CommitRecipe();
IF _recipePrepared THEN
    ParCfg := _parCfgStaged;
    // §8.11 performance references follow the model: OEE Performance denominator
    // and the WORK-time degradation baseline are per-recipe engineering data.
    Oee.IdealCycleMs := ParCfg.IdealCycleMs;
    Profiler.M_SetBaselineWork(WorkMs := ParCfg.BaselineWorkMs);
END_IF
_recipePrepared := FALSE;
END_METHOD

METHOD AbortRecipe
SUPER^.AbortRecipe();
_recipePrepared := FALSE;
END_METHOD

// First operational scan: initialize application-owned mode-chain state.
METHOD PROTECTED OnInit : DINT
OnInit := SUPER^.OnInit();
_M_ResetModeSequences();
_M_ClearModeTransitionState();
END_METHOD

// Every accepted Unit Start gets a fresh mode chain, including a repeated
// HOME/CHANGEOVER run that does not pass through another mode change.
METHOD PROTECTED OnCommandStart : DINT
OnCommandStart := SUPER^.OnCommandStart();
_M_ResetModeSequences();
END_METHOD

// Mode-entry wiring only. Step behavior remains in the selected sequence POU.
METHOD PROTECTED OnModeChanged : DINT
VAR_INPUT
    NewMode : E_Mode;
    OldMode : E_Mode;
END_VAR
OnModeChanged := SUPER^.OnModeChanged(
    NewMode := NewMode, OldMode := OldMode);
_M_ResetModeSequences();
_M_ClearModeTransitionState();
END_METHOD

METHOD PROTECTED OnCyclic : DINT
OnCyclic := SUPER^.OnCyclic();
// Project release engineering is a separate visible component. It owns the
// functional collision permits and mode-entry conditions consumed below.
ReleaseConditions.M_Evaluate(PressRam := PressRam, Door := Door, PartSlide := PartSlide,
    TwoHand := TwoHand, PneumaticPower := PneumaticPower,
    AirPressure := AirPressureMonitor);

// Latch access-gated Unit requests, then observe one full Execute-low scan before
// starting another power-group command (PLCopen edge discipline).
IF ControlOffRequest THEN
    _powerTargetOn := FALSE;
    _powerRequestPending := TRUE;
ELSIF ControlOnRequest THEN
    _powerTargetOn := TRUE;
    _powerRequestPending := TRUE;
END_IF
IF PneumaticPower.Done OR PneumaticPower.Error OR PneumaticPower.Aborted THEN
    PneumaticPower.Execute := FALSE;
ELSIF _powerRequestPending AND NOT PneumaticPower.Execute
AND (PneumaticPower.State = E_ExecState.READY) THEN
    PneumaticPower.Abort := FALSE;
    IF _powerTargetOn THEN
        PneumaticPower.Command := E_PowerGroupCommand.POWER_ON;
    ELSE
        PneumaticPower.Command := E_PowerGroupCommand.POWER_OFF;
    END_IF
    PneumaticPower.Execute := TRUE;
    _powerRequestPending := FALSE;
END_IF

// A physical two-hand edge may start AUTO from READY, or release an already
// running Unit's wait step. It never bypasses domain readiness or access policy.
IF TwoHand.OutImm.StartPulse
AND PartPresentSensor.OutImm.Value AND PartPresentSensor.OutImm.Quality
AND AirPressureMonitor.OutImm.PressureOk THEN
    IF (State = E_ExecState.BUSY) AND (ModeActive = E_Mode.AUTO) THEN
        _startLatched := TRUE;
    ELSIF (ModeActive = E_Mode.AUTO) AND Start() THEN
        _startLatched := TRUE;
    END_IF
ELSIF TwoHand.OutImm.StartPulse THEN
    _startLatched := FALSE;
END_IF
IF PneumaticPower.Error AND (State = E_ExecState.BUSY) THEN
    _M_RollupFault();
END_IF
IF (State = E_ExecState.BUSY)
AND NOT AirPressureMonitor.OutImm.PressureOk THEN
    PressRam.WithdrawOutputs();
    Door.WithdrawOutputs();
    PartSlide.WithdrawOutputs();
    _M_Fault(E_Reason.PERMISSIVE_NOT_MET, 'project.error.pressAirPressureLost');
END_IF
OutImm.PressRetracted := PressRam.OutImm.Retracted;
OutImm.DoorOpen := Door.OutImm.Retracted;
OutImm.DoorClosed := Door.OutImm.Extended;
OutImm.SlideInside := PartSlide.OutImm.Extended;
OutImm.SlideOutside := PartSlide.OutImm.Retracted;
OutImm.TwoHandArmed := TwoHand.OutImm.Armed;
OutImm.TwoHandActive := TwoHand.OutImm.SafeActive;
OutImm.PartPresent := PartPresentSensor.OutImm.Value AND PartPresentSensor.OutImm.Quality;
OutImm.AirPressureOk := AirPressureMonitor.OutImm.PressureOk;
OutImm.ReadyForLoad := Door.OutImm.Retracted AND NOT Door.OutImm.Extended
    AND PartSlide.OutImm.Retracted AND NOT PartSlide.OutImm.Extended
    AND PressRam.OutImm.Retracted AND NOT PressRam.OutImm.Extended;
OutImm.ActiveSettleTime := ParCfg.PressSettleTime;
OutImm.Diagnostic := Status.Diagnostic;
END_METHOD

METHOD PROTECTED OnAbort : DINT
OnAbort := SUPER^.OnAbort();
_M_PartAborted();                    // §3.16.3: the part leaves without a valid result
_M_WithdrawSequenceOutputs();
_M_ResetModeSequences();
_M_ClearModeTransitionState();
_powerTargetOn := FALSE;
_powerRequestPending := TRUE;
END_METHOD

// Error-state Abort is a deliberate recovery action but does not clear ERROR.
METHOD PROTECTED OnAbortInError : DINT
OnAbortInError := SUPER^.OnAbortInError();
_M_WithdrawSequenceOutputs();
_M_ResetModeSequences();
_M_ClearModeTransitionState();
_powerTargetOn := FALSE;
_powerRequestPending := TRUE;
END_METHOD

// One safe-stop wiring point shared by normal and error-state abort transitions.
METHOD PROTECTED _M_WithdrawSequenceOutputs
PressRam.WithdrawOutputs();
Door.WithdrawOutputs();
PartSlide.WithdrawOutputs();
PressRam.Execute := FALSE;
Door.Execute := FALSE;
PartSlide.Execute := FALSE;
END_METHOD

// Reset application-owned chain plumbing at lifecycle transitions. The chains'
// N000/N999 steps remain the only owners of process initialization/completion.
METHOD PROTECTED _M_ResetModeSequences
_homeSequence.M_Reset();
_changeoverSequence.M_Reset();
_autoSequence.M_Reset();
END_METHOD

// Clear state that must not survive init, mode entry, or either abort path.
// OnCommandStart deliberately does not call this: a physical start pulse may have
// been latched one scan before the inherited Execute edge is consumed.
METHOD PROTECTED _M_ClearModeTransitionState
Decision.Prompt := '';
DecisionAnswer := 0;
_startLatched := FALSE;
END_METHOD

// Application-only seam for ordinary hardwired Control On/Off buttons.
// It is a method (not OPC UA data), so HMI writes still use the access-gated
// ReqControlOn/ReqControlOff contract. The power CM rechecks safety and health.
METHOD RequestLocalControl : BOOL
VAR_INPUT
    ControlOn : BOOL;
END_VAR
_powerTargetOn := ControlOn;
_powerRequestPending := TRUE;
RequestLocalControl := TRUE;
END_METHOD

// §3.4.2 — the press paces every motion boundary through _M_StepGate, so
// SINGLE_STEP and HOLD_TO_RUN are supported (NON-SAFETY pacing; interlocks
// and the certified safety layer are unaffected).
METHOD PROTECTED _M_SupportsRunStyle : BOOL
VAR_INPUT
    Style : E_RunStyle;
END_VAR
_M_SupportsRunStyle := (Style = E_RunStyle.CONTINUOUS)
    OR (Style = E_RunStyle.SINGLE_STEP) OR (Style = E_RunStyle.HOLD_TO_RUN);
END_METHOD

METHOD PROTECTED _M_Supports : BOOL
VAR_INPUT
    Mode : E_Mode;
END_VAR
_M_Supports := (Mode = E_Mode.AUTO) OR (Mode = E_Mode.MANUAL)
    OR (Mode = E_Mode.HOME) OR (Mode = E_Mode.CHANGEOVER);
END_METHOD

// Thin mode router. Each supported sequence is a named method in the Unit tree.
METHOD PROTECTED _M_Dispatch
CASE ModeActive OF
    E_Mode.AUTO:
        _M_SequenceAuto();
    E_Mode.HOME:
        _M_SequenceHome();
    E_Mode.CHANGEOVER:
        _M_SequenceChangeover();
    E_Mode.MANUAL:
        _M_Fault(E_Reason.UNSUPPORTED_COMMAND, 'project.error.pressManualHasNoSequence');
ELSE
    _M_Fault(E_Reason.UNSUPPORTED_COMMAND, 'project.error.pressModeHasNoSequence');
END_CASE
END_METHOD

// Wiring-only HOME adapter. OnCommandStart owns the reset edge; the sequence POU
// owns every process step and terminal action.
METHOD PROTECTED _M_SequenceHome
_homeSequence.M_Run();
END_METHOD

// Wiring-only CHANGEOVER adapter. The §6.8 chain owns model validation, safe
// positioning, the operator decision, and completion logic.
METHOD PROTECTED _M_SequenceChangeover
_changeoverSequence.M_Run();
END_METHOD

// Wiring-only AUTO adapter. Every production command, wait, timer, decision,
// traceability action, and transition lives in the §6.8 chain.
METHOD PROTECTED _M_SequenceAuto
_autoSequence.M_Run();
END_METHOD

METHOD PROTECTED _M_RouteManual : BOOL
VAR_INPUT
    TargetPath : STRING(255);
    Value : DINT;
END_VAR
_M_RouteManual := FALSE;
IF TargetPath = PressRam.Name THEN
    _M_RouteManual := PressRam.ManualCommand(Value := Value);
ELSIF TargetPath = Door.Name THEN
    _M_RouteManual := Door.ManualCommand(Value := Value);
ELSIF TargetPath = PartSlide.Name THEN
    _M_RouteManual := PartSlide.ManualCommand(Value := Value);
ELSE
    _M_RouteManual := FALSE;
END_IF
END_METHOD

// §7.8 mode-entry release owned by this Unit. The base Start method consumes the
// same report the HMI displays, so this condition cannot become explanation-only.
METHOD PROTECTED _M_AppendInterlocks
VAR_IN_OUT
    Report : ST_ReleaseReport;
END_VAR
ReleaseConditions.M_AppendStart(Report := Report);
END_METHOD

METHOD PROTECTED _M_AppendManualInterlocks
VAR_INPUT
    TargetPath : STRING(255);
    Value : DINT;
END_VAR
VAR_IN_OUT
    Report : ST_ReleaseReport;
END_VAR
ReleaseConditions.M_AppendManual(TargetPath := TargetPath, Value := Value,
    PressRam := PressRam, Door := Door, PartSlide := PartSlide, Report := Report);
END_METHOD

METHOD PROTECTED _M_PublishStatus
SUPER^._M_PublishStatus();
OutImm.Diagnostic := Status.Diagnostic;
END_METHOD

// §3.10.2 — base walk (Unit facets + all child modules), then the project-owned
// fieldbus topology identity: static members of GVL_PressFieldbus.Topology are
// OPC.UA.DA=0 and reach the HMI only through this manifest.
METHOD M_AppendConfig : BOOL
VAR_INPUT
    Pager : REFERENCE TO FB_ConfigPager;
END_VAR
M_AppendConfig := SUPER^.M_AppendConfig(Pager := Pager);
F_AppendTopologyConfig(Topology := GVL_PressFieldbus.Topology, Pager := Pager);
END_METHOD

END_FUNCTION_BLOCK

// ---- 00_System/MAIN.TcPOU
// Virtual-commissioning application for one pneumatic press Unit.
// IMPORTANT: the Safe* values below simulate TwinSAFE outputs only. A deployed
// machine maps certified E-stop/two-hand/guard/safe-valve results from TwinSAFE.
PROGRAM MAIN
VAR
    RecipeCatalog : FB_PressRecipeCatalog;
    PartCarrier : FB_LocalPartCarrier;    // §3.16.2 BY_POSITION identity + local result ring
    AccessUsers : FB_LocalAccessProvider; // §7.7 commissioning user/PIN table
    // TF6100 TMC-Filtered publication starts at the deployed root instance.
    // The marker is inherited by PneumaticPress's published child symbols.
    {attribute 'OPC.UA.DA' := '1'}
    PneumaticPress : FB_PressDemoUnit;
    IoCatalog : FB_PressIoCatalog;
    IoDriver : FB_PressIoDriver;
    ControlDomain : FB_PressControlDomain;
    OutputAuthority : FB_PressOutputAuthority;
    SimulationDriver : FB_PressSimulationDriver;
    PressHal, DoorHal, SlideHal : ST_CylinderHal;
    TwoHandHal : ST_TwoHandHal;
    PowerHal : ST_PowerGroupHal;
    PartPresentHal : ST_DigitalInputHal;
    AirPressureHal : ST_AirPressureHal;
    InitialModel : ST_ModelId;
    Plate : ST_Nameplate;
    Init : BOOL;
    // Read-only MIRRORS of the commissioning gates (see the VAR CONSTANT block).
    // They exist only so the gate state stays visible over ADS/OPC UA: the
    // compiler inlines constants, which may publish no symbol at all, and losing
    // that visibility would remove the fastest way to diagnose "no output moves".
    // They are reassigned from the constants every cycle and nothing reads them,
    // so writing one online is inert - the constant remains the only authority.
    UseSimulation : BOOL;
    ControlCircuitMappingConfirmed : BOOL;
    // §10.5.1 demand gate, written by the HMI while its fieldbus page is open.
    // FALSE parks the EtherCAT master scan (no ADS traffic for a view nobody is
    // watching); the last read states are held, never falsified.
    FieldbusViewActive : BOOL;

    // Simulation controls. E-stop is normally closed: TRUE = healthy circuit.
    SimEStopNc : BOOL := TRUE;
    SimControlOnButton : BOOL;
    SimControlOffButton : BOOL;
    SimLeftButton : BOOL;
    SimRightButton : BOOL;
    SimSafetyValveOk : BOOL := TRUE;
    SimFieldbusHealthy : BOOL := TRUE;
    SimPartPresent : BOOL := TRUE;
    SimAirPressureOk : BOOL := TRUE;
    SafeEStopOk : BOOL;
    SafeGuardClosed : BOOL;
    SafeTwoHandActive : BOOL;
    SafePneumaticPermit : BOOL;
    SafetyFieldbusHealthy : BOOL;
    StandardIoHealthy : BOOL;
    RawEStopHealthy : BOOL;
    LampsOn : BOOL;
    ControlOnEdge : R_TRIG;
    ControlOffEdge : R_TRIG;
    ControlOnAdopted : R_TRIG;   // rising edge of the relay chain's feedback
END_VAR
VAR CONSTANT
    // COMMISSIONING GATES - deliberately CONSTANT so they cannot be flipped
    // online. Defeating a gate must be a source change plus a download: a
    // reviewable, auditable act, not a live write from an HMI or ADS client.
    //
    // TRUE makes MAIN call M_ClearOutputs() every cycle, so no physical output
    // is ever energized while the simulation driver animates the plant.
    USE_SIMULATION : BOOL := FALSE;
    // FALSE makes M_WriteOutputs force _000K951_A1 and _000K911_A1 FALSE every
    // cycle. Control On then cannot energize, the hardwired N54 D2 relay chain
    // never closes, and NOTHING moves - even though the cylinder coils are
    // written unconditionally. Set TRUE only after verifying the K951/K911
    // electrical semantics on the cabinet; per N54 D2 SwitchControlOn and
    // EnableControlOn are distinct signals.
    CONTROL_CIRCUIT_MAPPING_CONFIRMED : BOOL := TRUE;
END_VAR

// Mirror the compile-time gates so they remain observable (see declaration).
UseSimulation := USE_SIMULATION;
ControlCircuitMappingConfirmed := CONTROL_CIRCUIT_MAPPING_CONFIRMED;

IF NOT Init THEN
    Init := TRUE;
    // Initial mechanically safe/load position: ram up, door open, slide outside.
    PressHal.RetractedFb := TRUE;
    DoorHal.RetractedFb := TRUE;
    SlideHal.RetractedFb := TRUE;
    RecipeCatalog.Setup(UnitRef := PneumaticPress);
    PneumaticPress.Setup(Name := 'PneumaticPress', PressHal := PressHal, DoorHal := DoorHal,
        SlideHal := SlideHal, TwoHandHal := TwoHandHal, PowerHal := PowerHal,
        PartPresentHal := PartPresentHal, AirPressureHal := AirPressureHal,
        Recipe := RecipeCatalog.Provider);
    IoDriver.Setup(UnitRef := PneumaticPress);
    IoCatalog.Setup(UnitRef := PneumaticPress);
    ControlDomain.Setup(UnitRef := PneumaticPress);
    SimulationDriver.Setup(PressHal := PressHal, DoorHal := DoorHal, SlideHal := SlideHal);
    InitialModel.ModelCode := 'ALUMINUM';
    PneumaticPress.SetModel(Id := InitialModel);
    Plate.ProductUri := 'urn:fraktal:demo:pneumatic-press:2026-0001';
    Plate.ManufacturerName := 'Fraktal Example Project';
    Plate.ProductDesignation := 'Pneumatic Press Training Cell';
    Plate.SerialNumber := 'PRESS-DEMO-2026-0001';
    Plate.YearOfConstruction := '2026';
    Plate.SoftwareVersion := 'Fraktal Press Demo 0.1';
    PneumaticPress.SetNameplate(Plate := Plate);
    PneumaticPress.AlarmLog.RegisterMeta(Reason := E_Reason.INTERLOCK_DROPPED,
        OperatorAction := 'project.alarmAction.pressInterlock',
        Consequence := 'project.alarmConsequence.pressInterlock', Shelvable := FALSE);
    // §8.9 rationalization: per-reason operator action + consequence for the HMI join
    PneumaticPress.AlarmLog.RegisterMeta(Reason := E_Reason.PERMISSIVE_NOT_MET,
        OperatorAction := 'project.alarmAction.pressAirPressure',
        Consequence := 'project.alarmConsequence.pressAirPressure', Shelvable := FALSE);
    PneumaticPress.AlarmLog.RegisterMeta(Reason := E_Reason.RECIPE_INVALID,
        OperatorAction := 'project.alarmAction.pressRecipe',
        Consequence := 'project.alarmConsequence.pressRecipe', Shelvable := FALSE);
    PneumaticPress.AlarmLog.RegisterMeta(Reason := PL_ModuleReasons.CYL_WORK_NOT_REACHED,
        OperatorAction := 'project.alarmAction.pressCylinderPosition',
        Consequence := 'project.alarmConsequence.pressCylinderPosition', Shelvable := FALSE);
    PneumaticPress.AlarmLog.RegisterMeta(Reason := PL_ModuleReasons.CYL_HOME_NOT_REACHED,
        OperatorAction := 'project.alarmAction.pressCylinderPosition',
        Consequence := 'project.alarmConsequence.pressCylinderPosition', Shelvable := FALSE);
    // §3.16 traceability: station-local BY_POSITION serials; RFID/host substitutes later
    PartCarrier.Setup(UidPrefix := 'PRESS-2026-');
    PneumaticPress.SetPartCarrier(Carrier := PartCarrier);
    // §7.7 access: commissioning users (policy stays shipped-open; login is optional)
    AccessUsers.Register(User := 'operator', Pin := '1111', Level := E_AccessLevel.OPERATOR);
    AccessUsers.Register(User := 'tech', Pin := '2222', Level := E_AccessLevel.TECHNICIAN);
    AccessUsers.Register(User := 'admin', Pin := '9999', Level := E_AccessLevel.ADMIN);
    PneumaticPress.Access.Setup(Provider := AccessUsers, pAlarmLog := ADR(PneumaticPress.AlarmLog));
END_IF

// Ordinary simulated local station buttons. The worksheet does not list real
// Control On/Off input buttons; physical operation therefore uses HMI requests
// until those devices are identified. Control Off wins simultaneous edges.
// Source the Control On/Off edges from the REAL buttons on a live machine, and
// from the simulated ones only under USE_SIMULATION. Previously both edges were
// ANDed with USE_SIMULATION, so on hardware neither could ever fire and the
// machine had no headless Control On path at all.
IF USE_SIMULATION THEN
    ControlOnEdge(CLK := SimControlOnButton);
    ControlOffEdge(CLK := SimControlOffButton);
ELSE
    ControlOnEdge(CLK := IoDriver.ControlOnButton);
    ControlOffEdge(CLK := IoDriver.ControlOffButton);
END_IF
IF ControlOffEdge.Q THEN
    PneumaticPress.RequestLocalControl(ControlOn := FALSE);
ELSIF ControlOnEdge.Q THEN
    PneumaticPress.RequestLocalControl(ControlOn := TRUE);
END_IF
// Adopt the relay chain's established state: it is the authority. Without this
// the PLC can sit with no power request while K911_Y32 shows control is already
// ON (observed on the press), leaving PLC and hardware permanently out of step.
// One-shot: re-issuing POWER_ON every scan would re-fault the power group on
// any momentary permit dip and spam the event log. Latch on the feedback's
// rising edge only, and re-arm the latch when control drops away.
ControlOnAdopted(CLK := PowerHal.PowerFeedback);
IF NOT USE_SIMULATION AND ControlOnAdopted.Q AND NOT ControlOffEdge.Q THEN
    PneumaticPress.RequestLocalControl(ControlOn := TRUE);
END_IF

IF USE_SIMULATION THEN
    SimulationDriver.M_ReadInputs(DoorHal := DoorHal, TwoHandHal := TwoHandHal,
        PowerHal := PowerHal, PartPresentHal := PartPresentHal,
        AirPressureHal := AirPressureHal, RawEStopHealthy := RawEStopHealthy,
        SafeEStopOk := SafeEStopOk, SafeGuardClosed := SafeGuardClosed,
        SafeTwoHandActive := SafeTwoHandActive,
        SafePneumaticPermit := SafePneumaticPermit,
        SafetyFieldbusHealthy := SafetyFieldbusHealthy,
        StandardIoHealthy := StandardIoHealthy, SimEStopNc := SimEStopNc,
        SimLeftButton := SimLeftButton, SimRightButton := SimRightButton,
        SimSafetyValveOk := SimSafetyValveOk,
        SimFieldbusHealthy := SimFieldbusHealthy,
        SimPartPresent := SimPartPresent, SimAirPressureOk := SimAirPressureOk,
        PowerRequested := PowerHal.EnableRequestOut);
ELSE
    // The project Hardware Driver is the only raw process-image consumer.
    IoDriver.M_ReadInputs(PressHal := PressHal, DoorHal := DoorHal,
        SlideHal := SlideHal, TwoHandHal := TwoHandHal, PowerHal := PowerHal,
        PartPresentHal := PartPresentHal, AirPressureHal := AirPressureHal,
        RawEStopHealthy := RawEStopHealthy, SafeEStopOk := SafeEStopOk,
        SafeGuardClosed := SafeGuardClosed, SafeTwoHandActive := SafeTwoHandActive,
        SafePneumaticPermit := SafePneumaticPermit,
        SafetyFieldbusHealthy := SafetyFieldbusHealthy,
        StandardIoHealthy := StandardIoHealthy);
END_IF
TwoHandHal.SafeActive := SafeTwoHandActive;
TwoHandHal.FieldbusHealthy := SafetyFieldbusHealthy;
PowerHal.SafetyPermit := SafePneumaticPermit;
PowerHal.FieldbusHealthy := StandardIoHealthy;

ControlDomain.M_Update(SafeEStopOk := SafeEStopOk,
    SafeGuardClosed := SafeGuardClosed, SafeTwoHandActive := SafeTwoHandActive,
    SafePneumaticPermit := SafePneumaticPermit,
    SafetyFieldbusHealthy := SafetyFieldbusHealthy,
    StandardIoHealthy := StandardIoHealthy, RawEStopHealthy := RawEStopHealthy,
    PowerFeedback := PowerHal.PowerFeedback,
    PowerRequested := PowerHal.EnableRequestOut,
    TwoHandFieldbusHealthy := TwoHandHal.FieldbusHealthy);
PneumaticPress.ControlDomain := ControlDomain.Status;

// First execute ordinary control, then apply a standard-PLC withdrawal layer.
// This is defense in depth only: the real safety system owns pneumatic removal.
PneumaticPress();
OutputAuthority.M_Apply(PressHal := PressHal, DoorHal := DoorHal,
    SlideHal := SlideHal, PowerFeedback := PowerHal.PowerFeedback,
    SafePneumaticPermit := SafePneumaticPermit,
    StandardIoHealthy := StandardIoHealthy,
    HazardousRamPermit := SafeGuardClosed AND SafeTwoHandActive);
IF USE_SIMULATION THEN
    // Never leave physical outputs energized while virtual commissioning.
    IoDriver.M_ClearOutputs();
    SimulationDriver.M_RefreshPlant();
ELSE
    LampsOn := PneumaticPress.TwoHand.OutImm.Armed
        AND ControlDomain.Status.ReadyForStart
        AND PneumaticPress.OutImm.PartPresent AND PneumaticPress.OutImm.AirPressureOk;
    IoDriver.M_WriteOutputs(PressHal := PressHal, DoorHal := DoorHal,
        SlideHal := SlideHal, PowerHal := PowerHal, LampsOn := LampsOn,
        ControlCircuitMappingConfirmed := CONTROL_CIRCUIT_MAPPING_CONFIRMED);
END_IF
// Node state comes from the real EtherCAT master. §10.5.1 is a diagnostic
// surface, so the master is scanned only while a client is watching the bus
// view: the HMI sets FieldbusViewActive when its fieldbus page is open (the same
// on-demand gating the read tiers already apply to the topology data itself).
IoDriver.M_RefreshFieldbus(BusViewActive := FieldbusViewActive);

END_PROGRAM

// ---- 00_System/FB_PressIoDriver.TcPOU
// Project Hardware Driver layer. This is the only POU that accesses GVL_PressIO.
// It maps raw process-image symbols to semantic HALs and refreshes the Core
// topology publisher. It contains no sequence, mode, recipe or device behavior.
FUNCTION_BLOCK FB_PressIoDriver
VAR_OUTPUT
    // Raw N54 D2 operator buttons, republished so MAIN can drive Control On/Off
    // from hardware without becoming a second GVL_PressIO consumer.
    ControlOnButton  : BOOL;
    ControlOffButton : BOOL;
END_VAR
VAR
    _publisher : FB_IoTopologyPublisher;
    {attribute 'OPC.UA.DA' := '0'}
    _unit : REFERENCE TO FB_PressDemoUnit;
    _attached : BOOL;
    // Hardware Control-On adapter: reconstructs the safety-status mirrors from
    // the raw relay/sensor process image on a machine with a hardwired N54 D2
    // Control On circuit (no TwinSAFE controller). Status only; not a safety fn.
    _controlOn : FB_PressControlOnCircuit;
    // Reads the REAL EtherCAT slave states from the master and publishes each
    // node's live state — the fieldbus tree reflects hardware, not Control-On.
    _busHealth : FB_EcBusHealth;
END_VAR

;

METHOD Setup : BOOL
VAR_INPUT
    UnitRef : REFERENCE TO FB_PressDemoUnit;
END_VAR
VAR
    // Left all-zero: FB_EcBusHealth auto-detects the EtherCAT master's AmsNetId,
    // so the project needs no fieldbus address and no XAE link. Assign a value
    // here only for a non-standard master (remote, or several on one PC).
    ecMasterNetId : T_AmsNetIdArr;
END_VAR
_unit REF= UnitRef;
_attached := _publisher.Setup(DataRef := GVL_PressFieldbus.Topology, ResetData := FALSE)
    AND __ISVALIDREF(_unit);
// Map the press topology to the EtherCAT master's slaves. The catalog defines
// node 1 = CX2030 master, nodes 2..6 = the 5 EtherCAT slaves (EK1200 coupler,
// EL1809, EL2809, EL6001, EL9011) in master scan order.
_busHealth.Setup(Publisher := _publisher, MasterNetIdArr := ecMasterNetId,
    FirstSlaveNode := 2, SlaveCount := 5, MasterNodeIndex := 1);
Setup := _attached;
END_METHOD

METHOD M_ReadInputs
VAR_IN_OUT
    PressHal : ST_CylinderHal;
    DoorHal : ST_CylinderHal;
    SlideHal : ST_CylinderHal;
    TwoHandHal : ST_TwoHandHal;
    PowerHal : ST_PowerGroupHal;
    PartPresentHal : ST_DigitalInputHal;
    AirPressureHal : ST_AirPressureHal;
    RawEStopHealthy : BOOL;
    SafeEStopOk : BOOL;
    SafeGuardClosed : BOOL;
    SafeTwoHandActive : BOOL;
    SafePneumaticPermit : BOOL;
    SafetyFieldbusHealthy : BOOL;
    StandardIoHealthy : BOOL;
END_VAR
VAR
    // EtherCAT process-image validity, DETECTED from the fieldbus master by the
    // library (FB_EcBusHealth) — the project no longer declares/links a RealBusOk.
    busOk : BOOL;
END_VAR
busOk := _busHealth.M_BusOk();
// Physical feeder retracted = logical slide inside; extended = outside.
SlideHal.ExtendedFb := GVL_PressIO._101B301A;
SlideHal.RetractedFb := GVL_PressIO._101B301B;
DoorHal.ExtendedFb := GVL_PressIO._101B201A;
DoorHal.RetractedFb := GVL_PressIO._101B201B;
PressHal.ExtendedFb := GVL_PressIO._101B202A;
PressHal.RetractedFb := GVL_PressIO._101B202B;
TwoHandHal.RightPressed := GVL_PressIO._101S101;
TwoHandHal.LeftPressed := GVL_PressIO._101S102;
PartPresentHal.Value := GVL_PressIO._101B601;
AirPressureHal.LowPressure := GVL_PressIO._000MB085A_2;
AirPressureHal.OperatingPressure := GVL_PressIO._000MB085A_4;
PowerHal.PowerFeedback := GVL_PressIO._000K911_Y32;
// This machine's safety is a hardwired N54 D2 Control On relay chain, not a
// TwinSAFE controller, so the GVL_PressSafety AT %I* aliases are never written.
// Reconstruct the read-only safety-status mirrors from the raw relay/sensor
// process image via the Control-On adapter. The relay chain remains the safety
// authority; these values drive HMI/interlock display only.
_controlOn.M_Evaluate(
    // POLARITY: =000+S1-K910A:14 is "Emergency Switch 1 PRESSED" (N54 D2), and on
    // THIS machine the contact is CONFIRMED NORMALLY OPEN - not pressed reads
    // FALSE, pressed reads TRUE - so inverting it yields the "healthy" mirror
    // this adapter publishes. Read un-inverted, a healthy machine reported
    // E-stop-unhealthy and control power was withheld (POWER_ENABLE_WITHHELD)
    // even with the relay chain demonstrably closed.
    //
    // DEMO WIRING ONLY - NOT FAIL-SAFE. A normally-open E-stop contact cannot
    // distinguish "not pressed" from a broken wire, a pulled terminal or a dead
    // input card: all read FALSE, and this mirror would then report HEALTHY.
    // ISO 13850 / EN 60204-1 require a normally-CLOSED contact so that any break
    // forces the stop. A production machine must rewire to NC and drop this
    // inversion. This mirror is diagnostic only - the hardwired relay chain
    // remains the safety authority (Core Sec.9), which is what keeps the
    // non-fail-safe wiring tolerable on a demo rig and nowhere else.
    EStopHealthyMirror := NOT GVL_PressIO._000K910A,
    DoorClosed := GVL_PressIO._101B201A,
    LeftButton := GVL_PressIO._101S102,
    RightButton := GVL_PressIO._101S101,
    ControlOnFeedback := GVL_PressIO._000K911_Y32,
    BusOk := busOk,
    ControlOnButton := GVL_PressIO._000BS901,
    ControlOffButton := GVL_PressIO._000BS902,
    AirPressureOk := GVL_PressIO._000MB085A_4 AND NOT GVL_PressIO._000MB085A_2);
RawEStopHealthy := _controlOn.RawEStopHealthy;
SafeEStopOk := _controlOn.SafeEStopOk;
SafeGuardClosed := _controlOn.SafeGuardClosed;
SafeTwoHandActive := _controlOn.SafeTwoHandActive;
SafePneumaticPermit := _controlOn.SafePneumaticPermit;
SafetyFieldbusHealthy := _controlOn.SafetyFieldbusHealthy;
StandardIoHealthy := _controlOn.StandardIoHealthy;
PartPresentHal.Quality := StandardIoHealthy;
AirPressureHal.Quality := StandardIoHealthy;
ControlOnButton := GVL_PressIO._000BS901;
ControlOffButton := GVL_PressIO._000BS902;
END_METHOD

METHOD M_ClearOutputs
GVL_PressIO._101K301A := FALSE; GVL_PressIO._101K301B := FALSE;
GVL_PressIO._101K201A := FALSE; GVL_PressIO._101K201B := FALSE;
GVL_PressIO._101K202A := FALSE; GVL_PressIO._101K202B := FALSE;
GVL_PressIO._101P101 := FALSE; GVL_PressIO._101P102 := FALSE;
GVL_PressIO._000K951_A1 := FALSE; GVL_PressIO._000K911_A1 := FALSE;
END_METHOD

METHOD M_WriteOutputs
VAR_INPUT
    PressHal : ST_CylinderHal;
    DoorHal : ST_CylinderHal;
    SlideHal : ST_CylinderHal;
    PowerHal : ST_PowerGroupHal;
    LampsOn : BOOL;
    ControlCircuitMappingConfirmed : BOOL;
END_VAR
GVL_PressIO._101K301A := SlideHal.ExtendOut;
GVL_PressIO._101K301B := SlideHal.RetractOut;
GVL_PressIO._101K201A := DoorHal.ExtendOut;
GVL_PressIO._101K201B := DoorHal.RetractOut;
GVL_PressIO._101K202A := PressHal.ExtendOut;
GVL_PressIO._101K202B := PressHal.RetractOut;
GVL_PressIO._101P101 := LampsOn;
GVL_PressIO._101P102 := LampsOn;
IF ControlCircuitMappingConfirmed THEN
    // N54 D2: these are DIFFERENT signals. SwitchControlOn is the momentary
    // button coil (2 s pulse); EnableControlOn is the bus/air permissive that
    // must be TRUE whenever the machine is healthy. Driving both from one power
    // request was why the control circuit could never energize.
    GVL_PressIO._000K951_A1 := _controlOn.SwitchControlOn;
    GVL_PressIO._000K911_A1 := _controlOn.EnableControlOn;
ELSE
    GVL_PressIO._000K951_A1 := FALSE;
    GVL_PressIO._000K911_A1 := FALSE;
END_IF
END_METHOD

// Node state now comes from the REAL EtherCAT master (FB_EcBusHealth), NOT from
// the Control-On / StandardIoHealthy verdict — the HMI fieldbus tree mirrors
// the actual bus (as XAE shows it). StandardIoHealthy is no longer an input.
METHOD M_RefreshFieldbus
VAR_INPUT
    // §10.5.1: the bus picture is a diagnostic surface, so the master is only
    // scanned while a consumer is actually reading it (the HMI fieldbus view is
    // open). Pass FALSE to park the scan; published states are then held, not
    // invalidated. One scan always runs after Setup so M_BusOk() has real data.
    BusViewActive : BOOL;
END_VAR
VAR
    D : ST_Diagnostic;
END_VAR
IF _attached THEN
    _busHealth.M_RequestScan(Active := BusViewActive);
    _busHealth.M_Refresh();  // publishes each node's real INIT/PREOP/SAFEOP/OP/FAULT
    _publisher.M_SetDigitalValue(NodeIndex := 3, ChannelIndex := 1, Value := GVL_PressIO._101B301A);
    _publisher.M_SetDigitalValue(NodeIndex := 3, ChannelIndex := 2, Value := GVL_PressIO._101B301B);
    _publisher.M_SetDigitalValue(NodeIndex := 3, ChannelIndex := 3, Value := GVL_PressIO._101B201A);
    _publisher.M_SetDigitalValue(NodeIndex := 3, ChannelIndex := 4, Value := GVL_PressIO._101B201B);
    _publisher.M_SetDigitalValue(NodeIndex := 3, ChannelIndex := 5, Value := GVL_PressIO._101B202A);
    _publisher.M_SetDigitalValue(NodeIndex := 3, ChannelIndex := 6, Value := GVL_PressIO._101B202B);
    _publisher.M_SetDigitalValue(NodeIndex := 3, ChannelIndex := 7, Value := GVL_PressIO._101S101);
    _publisher.M_SetDigitalValue(NodeIndex := 3, ChannelIndex := 8, Value := GVL_PressIO._101S102);
    _publisher.M_SetDigitalValue(NodeIndex := 3, ChannelIndex := 9, Value := GVL_PressIO._000MB085A_2);
    _publisher.M_SetDigitalValue(NodeIndex := 3, ChannelIndex := 10, Value := GVL_PressIO._000MB085A_4);
    _publisher.M_SetDigitalValue(NodeIndex := 3, ChannelIndex := 11, Value := GVL_PressIO._101B601);
    _publisher.M_SetDigitalValue(NodeIndex := 3, ChannelIndex := 12, Value := GVL_PressIO._000K911_Y32);
    _publisher.M_SetDigitalValue(NodeIndex := 3, ChannelIndex := 13, Value := GVL_PressIO._000K910A);
    _publisher.M_SetDigitalValue(NodeIndex := 4, ChannelIndex := 1, Value := GVL_PressIO._101K301A);
    _publisher.M_SetDigitalValue(NodeIndex := 4, ChannelIndex := 2, Value := GVL_PressIO._101K301B);
    _publisher.M_SetDigitalValue(NodeIndex := 4, ChannelIndex := 3, Value := GVL_PressIO._101K201A);
    _publisher.M_SetDigitalValue(NodeIndex := 4, ChannelIndex := 4, Value := GVL_PressIO._101K201B);
    _publisher.M_SetDigitalValue(NodeIndex := 4, ChannelIndex := 5, Value := GVL_PressIO._101K202A);
    _publisher.M_SetDigitalValue(NodeIndex := 4, ChannelIndex := 6, Value := GVL_PressIO._101K202B);
    _publisher.M_SetDigitalValue(NodeIndex := 4, ChannelIndex := 7, Value := GVL_PressIO._101P101);
    _publisher.M_SetDigitalValue(NodeIndex := 4, ChannelIndex := 8, Value := GVL_PressIO._101P102);
    _publisher.M_SetDigitalValue(NodeIndex := 4, ChannelIndex := 9, Value := GVL_PressIO._000K951_A1);
    _publisher.M_SetDigitalValue(NodeIndex := 4, ChannelIndex := 10, Value := GVL_PressIO._000K911_A1);
    _publisher.M_BeginDiagnosticRefresh();
    D := _unit.PressRam.Status.Diagnostic;
    _M_ApplyCylinderDiagnostic(Diagnostic := D,
        ExtendedTag := _unit.PressRam.OutImm.ExtendedSensorTag,
        RetractedTag := _unit.PressRam.OutImm.RetractedSensorTag);
    D := _unit.Door.Status.Diagnostic;
    _M_ApplyCylinderDiagnostic(Diagnostic := D,
        ExtendedTag := _unit.Door.OutImm.ExtendedSensorTag,
        RetractedTag := _unit.Door.OutImm.RetractedSensorTag);
    D := _unit.PartSlide.Status.Diagnostic;
    _M_ApplyCylinderDiagnostic(Diagnostic := D,
        ExtendedTag := _unit.PartSlide.OutImm.ExtendedSensorTag,
        RetractedTag := _unit.PartSlide.OutImm.RetractedSensorTag);
    D := _unit.AirPressureMonitor.Status.Diagnostic;
    _publisher.M_ApplyDiagnostic(Diagnostic := D);
    IF TO_DINT(D.ReasonCode) = PL_ModuleReasons.AIR_SWITCH_CONFLICT THEN
        _publisher.M_ApplyDiagnosticToTag(Diagnostic := D,
            Tag := _unit.AirPressureMonitor.OutImm.LowSensorTag);
        _publisher.M_ApplyDiagnosticToTag(Diagnostic := D,
            Tag := _unit.AirPressureMonitor.OutImm.OperatingSensorTag);
    ELSE
        ;
    END_IF
    _publisher.M_ApplyDiagnostic(Diagnostic := _unit.Status.Diagnostic);
ELSE
    ;
END_IF
END_METHOD

METHOD PRIVATE _M_ApplyCylinderDiagnostic
VAR_INPUT
    Diagnostic : ST_Diagnostic;
    ExtendedTag : STRING(80);
    RetractedTag : STRING(80);
END_VAR
_publisher.M_ApplyDiagnostic(Diagnostic := Diagnostic);
IF TO_DINT(Diagnostic.ReasonCode) = PL_ModuleReasons.CYL_BOTH_SENSORS THEN
    _publisher.M_ApplyDiagnosticToTag(Diagnostic := Diagnostic, Tag := ExtendedTag);
    _publisher.M_ApplyDiagnosticToTag(Diagnostic := Diagnostic, Tag := RetractedTag);
ELSE
    ;
END_IF
END_METHOD

END_FUNCTION_BLOCK

// ---- 00_System/FB_PressControlOnCircuit.TcPOU
// Hardware Control-On adapter for a machine whose safety is a HARDWIRED relay
// chain (Bosch/Nexeed N54 D2 "Control On", Pilz-style), NOT a TwinSAFE
// controller. The standard PLC is not a safety function here: the relay circuit
// remains the safety authority. This adapter only RECONSTRUCTS the read-only
// GVL_PressSafety-equivalent status the rest of the application expects, from the
// ordinary process-image inputs and the relay-chain Control On feedback, so the
// HMI and interlocks reflect the real machine instead of failing closed on
// unlinked TwinSAFE aliases.
//
// It produces status only (no safe outputs). The functional EnableControlOn /
// SwitchControlOn requests to the relay chain are driven by the existing power
// group -> FB_PressIoDriver.M_WriteOutputs path, gated by
// ControlCircuitMappingConfirmed until the electrical semantics are confirmed.
FUNCTION_BLOCK FB_PressControlOnCircuit
VAR_OUTPUT
    // Read-only mirrors, matching the six GVL_PressSafety aliases + the raw
    // E-stop mirror the driver forwards. TRUE = healthy/safe/present.
    RawEStopHealthy       : BOOL;
    SafeEStopOk           : BOOL;
    SafeGuardClosed       : BOOL;
    SafeTwoHandActive     : BOOL;
    SafePneumaticPermit   : BOOL;
    SafetyFieldbusHealthy : BOOL;
    StandardIoHealthy     : BOOL;
END_VAR

;

// Reconstruct the status mirrors from raw relay/sensor inputs. All inputs are
// ordinary (non-safety-rated) process-image values; the relay chain owns the
// actual safety function. Called once per scan by FB_PressIoDriver, the sole
// GVL_PressIO consumer.
METHOD M_Evaluate
VAR_INPUT
    EStopHealthyMirror : BOOL; // _000K910A: ordinary E-stop-healthy mirror
    DoorClosed         : BOOL; // _101B201A: guard-door closed sensor
    LeftButton         : BOOL; // _101S102: left two-hand raw button
    RightButton        : BOOL; // _101S101: right two-hand raw button
    ControlOnFeedback  : BOOL; // _000K911_Y32: relay-chain Control On established
    BusOk              : BOOL; // EtherCAT process image valid (link master OP state)
END_VAR
// Fieldbus health: the standard and (functional) safety I/O share one EtherCAT
// segment on this machine, so both mirror the bus-valid signal.
StandardIoHealthy     := BusOk;
SafetyFieldbusHealthy := BusOk;

// E-stop: the ordinary healthy mirror gated by a valid process image. This is a
// diagnostic mirror of the relay-chain E-stop, not an evaluated safe result.
RawEStopHealthy := EStopHealthyMirror;
SafeEStopOk     := EStopHealthyMirror AND BusOk;

// Guard: the door-closed sensor. Plausibility (per N54 D2 Safety Door add-on) is
// enforced in the relay chain; here it is the single available door signal.
SafeGuardClosed := DoorClosed AND BusOk;

// Two-hand: functional (both raw buttons) with E-stop healthy. The safety-rated
// two-hand evaluation lives in the relay chain; this drives interlock/HMI only.
SafeTwoHandActive := LeftButton AND RightButton AND SafeEStopOk AND BusOk;

// Pneumatic permit: the relay-chain Control On feedback IS the enabled state.
// Per N54 D2 the Main/Safety Valve add-ons already reset EnableControlOn on a
// compressed-air error and the Safety Door add-on on a guard error, so the
// K911_Y32 feedback subsumes air + guard monitoring. Gate on E-stop for defense
// in depth (the air-pressure inputs are read separately by the air HAL).
SafePneumaticPermit := ControlOnFeedback AND SafeEStopOk;
END_METHOD

END_FUNCTION_BLOCK

// ---- 00_System/FB_PressControlDomain.TcPOU
// Application control-domain coordinator (Core §9.8). It describes one cage and
// pneumatic power arrangement; it is infrastructure, not a fourth module tier.
FUNCTION_BLOCK FB_PressControlDomain
VAR_OUTPUT
    Status : ST_ControlDomainStatus;
END_VAR
VAR
    {attribute 'OPC.UA.DA' := '0'}
    _unit : REFERENCE TO FB_PressDemoUnit;
    _attached : BOOL;
END_VAR

;

METHOD Setup : BOOL
VAR_INPUT
    UnitRef : REFERENCE TO FB_PressDemoUnit;
END_VAR
_unit REF= UnitRef;
_attached := __ISVALIDREF(_unit);
Status.Present := TRUE;
Status.Id := 'PRESS-CAGE-01';
Status.Name := 'project.controlDomain.press.name';
Status.MemberCount := 1;
Status.MemberUnitPaths[1] := UnitRef.Name;
Status.Safety.Present := TRUE;
Status.Safety.DeviceCount := 4;
Status.Safety.Devices[1].Present := TRUE;
Status.Safety.Devices[1].Name := 'EStop01';
Status.Safety.Devices[1].Kind := E_SafetyDeviceKind.ESTOP;
Status.Safety.Devices[1].AffectedPowerMask := 16#0000_0001;
Status.Safety.Devices[1].Description := 'project.safety.estopNc';
Status.Safety.Devices[2].Present := TRUE;
Status.Safety.Devices[2].Name := 'PressGuard';
Status.Safety.Devices[2].Kind := E_SafetyDeviceKind.GUARD_DOOR;
Status.Safety.Devices[2].AffectedPowerMask := 16#0000_0001;
Status.Safety.Devices[2].Description := 'project.safety.pressGuard';
Status.Safety.Devices[3].Present := TRUE;
Status.Safety.Devices[3].Name := 'TwoHand01';
Status.Safety.Devices[3].Kind := E_SafetyDeviceKind.TWO_HAND_CONTROL;
Status.Safety.Devices[3].AffectedPowerMask := 16#0000_0001;
Status.Safety.Devices[3].Description := 'project.safety.twoHandControl';
Status.Safety.Devices[4].Present := TRUE;
Status.Safety.Devices[4].Name := 'SafeValve01';
Status.Safety.Devices[4].Kind := E_SafetyDeviceKind.SAFETY_VALVE;
Status.Safety.Devices[4].AffectedPowerMask := 16#0000_0001;
Status.Safety.Devices[4].Description := 'project.safety.pressSafeValve';
Status.ControlPower.Present := TRUE;
Status.ControlPower.GroupCount := 1;
Setup := _attached;
END_METHOD

METHOD M_Update
VAR_INPUT
    SafeEStopOk : BOOL;
    SafeGuardClosed : BOOL;
    SafeTwoHandActive : BOOL;
    SafePneumaticPermit : BOOL;
    SafetyFieldbusHealthy : BOOL;
    StandardIoHealthy : BOOL;
    RawEStopHealthy : BOOL;
    PowerFeedback : BOOL;
    PowerRequested : BOOL;
    TwoHandFieldbusHealthy : BOOL;
END_VAR
IF _attached THEN
    Status.Safety.AllSafe := SafeEStopOk AND SafePneumaticPermit AND SafetyFieldbusHealthy;
    Status.Safety.DemandActive := NOT SafeGuardClosed;
    Status.Safety.ResetRequired := NOT SafeEStopOk;
    Status.Safety.FaultActive := NOT SafetyFieldbusHealthy OR NOT StandardIoHealthy
        OR (RawEStopHealthy <> SafeEStopOk);
    Status.Safety.Devices[1].State := SEL(SafeEStopOk, E_SafetyState.DEMAND, E_SafetyState.READY);
    Status.Safety.Devices[1].Ready := SafeEStopOk;
    Status.Safety.Devices[1].DemandActive := NOT SafeEStopOk;
    Status.Safety.Devices[1].SafeStateActive := NOT SafeEStopOk;
    Status.Safety.Devices[1].ResetRequired := NOT SafeEStopOk;
    Status.Safety.Devices[1].FieldbusHealthy := SafetyFieldbusHealthy;
    Status.Safety.Devices[2].State := SEL(SafeGuardClosed, E_SafetyState.SAFE_STATE, E_SafetyState.READY);
    Status.Safety.Devices[2].Ready := SafeGuardClosed;
    Status.Safety.Devices[2].DemandActive := NOT SafeGuardClosed;
    Status.Safety.Devices[2].SafeStateActive := NOT SafeGuardClosed;
    Status.Safety.Devices[2].FieldbusHealthy := SafetyFieldbusHealthy;
    Status.Safety.Devices[3].State := SEL(SafeTwoHandActive, E_SafetyState.READY, E_SafetyState.DEMAND);
    Status.Safety.Devices[3].Ready := TwoHandFieldbusHealthy;
    Status.Safety.Devices[3].DemandActive := SafeTwoHandActive;
    Status.Safety.Devices[3].SafeStateActive := NOT SafeTwoHandActive;
    Status.Safety.Devices[3].FieldbusHealthy := SafetyFieldbusHealthy;
    Status.Safety.Devices[4].State := SEL(SafePneumaticPermit, E_SafetyState.FAULT, E_SafetyState.READY);
    Status.Safety.Devices[4].Ready := SafePneumaticPermit;
    Status.Safety.Devices[4].DemandActive := NOT SafePneumaticPermit;
    Status.Safety.Devices[4].SafeStateActive := NOT SafePneumaticPermit;
    Status.Safety.Devices[4].FaultActive := NOT SafePneumaticPermit;
    Status.Safety.Devices[4].FieldbusHealthy := SafetyFieldbusHealthy;
    Status.ControlPower.RequestedOn := PowerRequested;
    Status.ControlPower.ControlOn := PowerFeedback;
    Status.ControlPower.Transitioning := _unit.PneumaticPower.Busy;
    Status.ControlPower.RearmRequired := _unit.PneumaticPower.ControlPower.RearmRequired;
    Status.ControlPower.Groups[1] := _unit.PneumaticPower.OutImm.Status;
    Status.ReadyForStart := Status.Safety.AllSafe AND Status.ControlPower.ControlOn
        AND NOT Status.ControlPower.RearmRequired;
ELSE
    Status.ReadyForStart := FALSE;
END_IF
END_METHOD

END_FUNCTION_BLOCK
